FUNCTION_BLOCK PUBL_1_COMM (* 2-variable data publisher *)
  (* Standard: 61499-2 *)
  (* Version 1.0, 21-03-12, GASR, Universidade do Estado de Santa Catarina *)
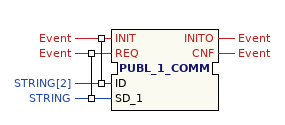
  EVENT_INPUT
    INIT WITH ID; (* Service initiaization *)
    REQ WITH SD_1;
  END_EVENT
  EVENT_OUTPUT
    INITO; (* Initialization Confirm *)
    CNF; (* Service confirmation *)
  END_EVENT
  VAR_INPUT
    ID : ARRAY [0..1] OF STRING; (* Default id is the FB instance name *)
    SD_1 : STRING; (* Filename *)
  END_VAR
  SERVICE PUBL_1/SUBL_1 (* Data publication service *)
    SEQUENCE normal_establishment
      PUBL_1.INIT(ID) -> PUBL_1.INITO();
      SUBL_1.INIT(ID) -> SUBL_1.INITO();
    END_SEQUENCE
    SEQUENCE normal_data_transfer
      PUBL_1.REQ(SD_1) -> Subl_1.IND(RD_1);
    END_SEQUENCE
  END_SERVICE
END_FUNCTION_BLOCK
